// TIA Portal V16 export
// export: Created 2021-07-12T14:47:18.4549797Z, ExportSetting WithDefaults, DisplayName Totally Integrated Automation Portal, DisplayVersion V16, DisplayName TIA Portal Version Control Interface, DisplayVersion V16, DisplayName TIA Portal Openness, DisplayVersion V16, DisplayName STEP 7 Professional, DisplayVersion V16, DisplayName STEP 7 Safety, DisplayVersion V16, DisplayName WinCC Professional, DisplayVersion V16
TYPE "LSimaHydTO_typeStatusTransducer"
TITLE = LSimaHydTO_typeStatusTransducer
// Indicates the status of transducer data
// stored: IsFailsafeCompliant false
   STRUCT
      RawValue : Word;   // Raw data of analog input
      PressureValue : LReal;   // actual pressure In pressure units
      ForceValue : LReal;   // actual force In force units
      Error : Bool := FALSE;   // Indicates error of transducer
   END_STRUCT;
END_TYPE
